FUNCTION_BLOCK FB_SimpleLinearTwoWayDrive_Test EXTENDS FB_TestSuite
VAR_INPUT
END_VAR
VAR_OUTPUT
END_VAR
VAR
END_VAR

METHOD No_Movement_When_Locked : BOOL
VAR_INPUT
END_VAR
VAR
	sut: FB_SimpleLinearTwoWayDrive;
END_VAR
TEST('No movement should be possible when locked');

sut(
	SensorHomePos := TRUE,
	SensorWorkPos := FALSE,
	Enable := FALSE,
	ToHome := FALSE,
	ToWork := FALSE);
	
AssertEquals(FALSE, sut.ActorWorkPos, 'Movement even if not enabled');

TEST_FINISHED();
END_METHOD

END_FUNCTION_BLOCK

(* stored: Version 1.1.0.1, ProductVersion 3.1.4024.11
   POU FB_SimpleLinearTwoWayDrive_Test: Id {d9e1087f-58a6-4e65-903c-24417411064b}, SpecialFunc None
   Method No_Movement_When_Locked: Id {74abaccd-090b-4cac-b60e-cf51473bfb80} *)
